FUNCTION_BLOCK PICKER_VIEW_NEW (* View Composite FB *)
  (* Standard: 61499-2 *)
  (* Version 0.2, 2003-12-05, JHC, Rockwell Automation, Renamed from NEWCOMPFB. *)
  (* Version 0.1, 2002-01-08, JHC, Rockwell Automation, Added DLY FB as example. *)
  (* Version 0.0, 2000-05-27, JHC, Rockwell Automation *)
  (* Compiler header: package fb.rt.pnp;import fb.rt.vhmi.*;import fb.rt.math.*;import fb.rt.vmath.*; *)
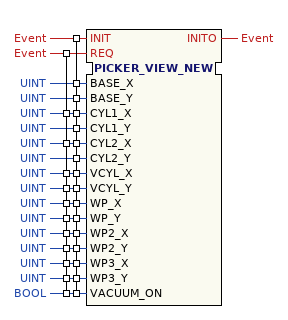
  EVENT_INPUT
    INIT WITH BASE_X, BASE_Y, CYL1_Y, CYL2_Y, CYL1_X, CYL2_X, VCYL_X, VCYL_Y, WP_X, WP_Y, VACUUM_ON, WP2_Y, WP2_X, WP3_X, WP3_Y; (* Initialization Request *)
    REQ WITH CYL1_X, CYL2_X, VCYL_X, VCYL_Y, WP_X, WP_Y, VACUUM_ON, WP2_X, WP2_Y, WP3_X, WP3_Y; (* Normal Execution Request *)
  END_EVENT
  EVENT_OUTPUT
    INITO; (* Initialization Confirm *)
  END_EVENT
  VAR_INPUT
    BASE_X : UINT;
    BASE_Y : UINT;
    CYL1_X : UINT;
    CYL1_Y : UINT;
    CYL2_X : UINT;
    CYL2_Y : UINT;
    VCYL_X : UINT;
    VCYL_Y : UINT;
    WP_X : UINT;
    WP_Y : UINT;
    WP2_X : UINT;
    WP2_Y : UINT;
    WP3_X : UINT;
    WP3_Y : UINT;
    VACUUM_ON : BOOL;
  END_VAR
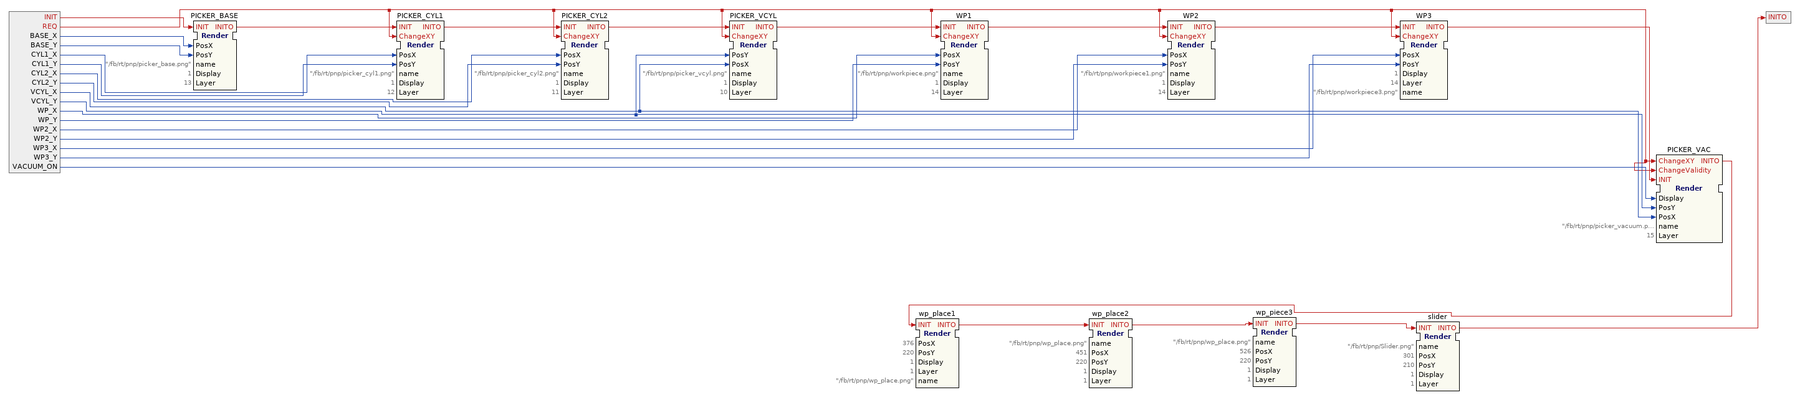
  FBS
    PICKER_BASE : Render(name := "/fb/rt/pnp/picker_base.png", Display := 1, Layer := 13);
    PICKER_CYL1 : Render(name := "/fb/rt/pnp/picker_cyl1.png", Display := 1, Layer := 12);
    PICKER_CYL2 : Render(name := "/fb/rt/pnp/picker_cyl2.png", Display := 1, Layer := 11);
    PICKER_VCYL : Render(name := "/fb/rt/pnp/picker_vcyl.png", Display := 1, Layer := 10);
    WP1 : Render(name := "/fb/rt/pnp/workpiece.png", Display := 1, Layer := 14);
    PICKER_VAC : Render(name := "/fb/rt/pnp/picker_vacuum.png", Layer := 15);
    wp_place1 : Render(PosX := 376, PosY := 220, Display := 1, Layer := 1, name := "/fb/rt/pnp/wp_place.png");
    wp_place2 : Render(name := "/fb/rt/pnp/wp_place.png", PosX := 451, PosY := 220, Display := 1, Layer := 1);
    wp_piece3 : Render(name := "/fb/rt/pnp/wp_place.png", PosX := 526, PosY := 220, Display := 1, Layer := 1);
    slider : Render(name := "/fb/rt/pnp/Slider.png", PosX := 301, PosY := 210, Display := 1, Layer := 1);
    WP2 : Render(name := "/fb/rt/pnp/workpiece1.png", Display := 1, Layer := 14);
    WP3 : Render(Display := 1, Layer := 14, name := "/fb/rt/pnp/workpiece3.png");
  END_FBS
  EVENT_CONNECTIONS
    INIT TO PICKER_BASE.INIT;
    PICKER_BASE.INITO TO PICKER_CYL1.INIT;
    PICKER_CYL1.INITO TO PICKER_CYL2.INIT;
    PICKER_CYL2.INITO TO PICKER_VCYL.INIT;
    PICKER_VCYL.INITO TO WP1.INIT;
    REQ TO PICKER_CYL1.ChangeXY;
    REQ TO PICKER_CYL2.ChangeXY;
    REQ TO PICKER_VCYL.ChangeXY;
    REQ TO WP1.ChangeXY;
    REQ TO PICKER_VAC.ChangeXY;
    REQ TO PICKER_VAC.ChangeValidity;
    wp_place1.INITO TO wp_place2.INIT;
    wp_place2.INITO TO wp_piece3.INIT;
    wp_piece3.INITO TO slider.INIT;
    WP1.INITO TO WP2.INIT;
    WP2.INITO TO WP3.INIT;
    WP3.INITO TO PICKER_VAC.INIT;
    REQ TO WP2.ChangeXY;
    REQ TO WP3.ChangeXY;
    PICKER_VAC.INITO TO wp_place1.INIT;
    slider.INITO TO INITO;
  END_CONNECTIONS
  DATA_CONNECTIONS
    VACUUM_ON TO PICKER_VAC.Display;
    BASE_X TO PICKER_BASE.PosX;
    BASE_Y TO PICKER_BASE.PosY;
    CYL1_X TO PICKER_CYL1.PosX;
    CYL2_X TO PICKER_CYL2.PosX;
    VCYL_Y TO PICKER_VCYL.PosY;
    WP_X TO WP1.PosX;
    WP_Y TO WP1.PosY;
    VCYL_Y TO PICKER_VAC.PosY;
    CYL1_Y TO PICKER_CYL1.PosY;
    VCYL_X TO PICKER_VCYL.PosX;
    VCYL_X TO PICKER_VAC.PosX;
    CYL2_Y TO PICKER_CYL2.PosY;
    WP2_X TO WP2.PosX;
    WP2_Y TO WP2.PosY;
    WP3_X TO WP3.PosX;
    WP3_Y TO WP3.PosY;
  END_CONNECTIONS
END_FUNCTION_BLOCK
